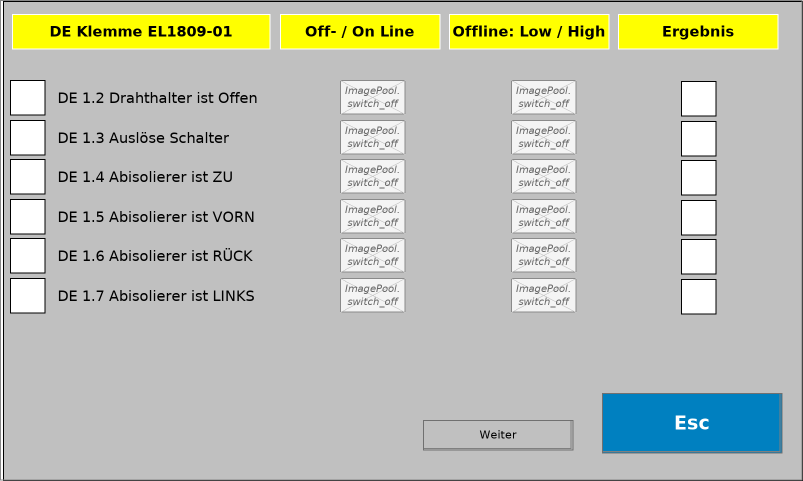
VISUALIZATION IO_Visu01  // 803x481
    Rectangle (3,1 800x480)
    Rectangle (12,14 258x35), "DE Klemme EL1809-01"
    Label (50,83 228x30), "DE 1.2 Drahthalter ist Offen"
    Label (50,123 201x30), "DE 1.3 Auslöse Schalter"
    Label (50,162 201x30), "DE 1.4 Abisolierer ist ZU"
    Label (50,202 233x30), "DE 1.5 Abisolierer ist VORN"
    Label (50,241 245x30), "DE 1.6 Abisolierer ist RÜCK"
    Rectangle (10,80 35x35), colour toggle: IO.inDrahthalterIstOffen
    Rectangle (10,120 35x35), colour toggle: IO.inAusloeseSchalter
    Rectangle (10,159 35x35), colour toggle: IO.inAbisoliererIstZU
    Rectangle (10,199 35x35), colour toggle: IO.inAbisoliererIstVORN
    Rectangle (10,238 35x35), colour toggle: IO.inAbisoliererIstRUECK
    Rectangle (10,278 35x35), colour toggle: IO.inAbisoliererIstLINKS
    Label (50,281 260x30), "DE 1.7 Abisolierer ist LINKS"
    Rectangle (280,14 160x35), "Off- / On Line"
    Image (340,80 65x34), image: ImagePool.switch_off
        p84334746: P_InputHandling.E1_2.onlineImageID
        OnMouseUp: execute { RVL.e12Online := NOT RVL.e12Online; }
    Image (340,120 65x34), image: ImagePool.switch_off
        p84334746: P_InputHandling.E1_3.onlineImageID
        OnMouseUp: execute { RVL.e13Online := NOT RVL.e13Online; }
    Image (340,159 65x34), image: ImagePool.switch_off
        p84334746: P_InputHandling.E1_4.onlineImageID
        OnMouseUp: execute { RVL.e14Online := NOT RVL.e14Online; }
    Image (340,199 65x34), image: ImagePool.switch_off
        p84334746: P_InputHandling.E1_5.onlineImageID
        OnMouseUp: execute { RVL.e15Online := NOT RVL.e15Online; }
    Image (340,238 65x34), image: ImagePool.switch_off
        p84334746: P_InputHandling.E1_6.onlineImageID
        OnMouseUp: execute { RVL.e16Online := NOT RVL.e16Online; }
    Image (340,278 65x34), image: ImagePool.switch_off
        p84334746: P_InputHandling.E1_7.onlineImageID
        OnMouseUp: execute { RVL.e17Online := NOT RVL.e17Online; }
    Rectangle (449,14 160x35), "Offline: Low / High"
    Image (511,80 65x34), image: ImagePool.switch_off
        p84334746: P_InputHandling.E1_2.modeImageID
        OnMouseUp: execute { RVL.e12OffMode := NOT RVL.e12OffMode; }
    Image (511,120 65x34), image: ImagePool.switch_off
        p84334746: P_InputHandling.E1_3.modeImageID
        OnMouseUp: execute { RVL.e13OffMode := NOT RVL.e13OffMode; }
    Image (511,159 65x34), image: ImagePool.switch_off
        p84334746: P_InputHandling.E1_4.modeImageID
        OnMouseUp: execute { RVL.e14OffMode := NOT RVL.e14OffMode; }
    Image (511,199 65x34), image: ImagePool.switch_off
        p84334746: P_InputHandling.E1_5.modeImageID
        OnMouseUp: execute { RVL.e15OffMode := NOT RVL.e15OffMode; }
    Image (511,238 65x34), image: ImagePool.switch_off
        p84334746: P_InputHandling.E1_6.modeImageID
        OnMouseUp: execute { RVL.e16OffMode := NOT RVL.e16OffMode; }
    Image (511,278 65x34), colour toggle: GVL.insecAbisoliererIstLINKS, image: ImagePool.switch_off
        p84334746: P_InputHandling.E1_7.modeImageID
        OnMouseUp: execute { RVL.e17OffMode := NOT RVL.e17OffMode; }
    Rectangle (681,81 35x35), colour toggle: GVL.insecDrahthalterIstOffen
    Rectangle (681,121 35x35), colour toggle: GVL.insecAusloeseSchalter
    Rectangle (681,160 35x35), colour toggle: GVL.insecAbisoliererIstZU
    Rectangle (681,200 35x35), colour toggle: GVL.insecAbisoliererIstVORN
    Rectangle (681,239 35x35), colour toggle: GVL.insecAbisoliererIstRUECK
    Rectangle (681,279 35x35), colour toggle: GVL.insecAbisoliererIstLINKS
    Rectangle (618,14 160x35), "Ergebnis"
    Button (423,420 150x30), "Weiter"
        OnMouseClick: change screen: IO_Visu02
    Button (602,393 180x60), "Esc"
        OnMouseUp: change screen: Menu
END_VISUALIZATION

(* stored: Version 1.1.0.1, ProductVersion 3.1.4024.3
   Visu IO_Visu01: Id {80fc96ba-6564-44bb-80f6-c87951262215} *)
